# EPICS substitutions: mc1/GalilTestApp/Db/galil_digital_ports.substitutions
# Description:
# digital/binary port substitution file.
#
# This library is free software; you can redistribute it and/or
# modify it under the terms of the GNU Lesser General Public
# Licence as published by the Free Software Foundation; either
# version 2.1 of the Licence, or (at your option) any later version.
#
# This library is distributed in the hope that it will be useful,
# but WITHOUT ANY WARRANTY; without even the implied warranty of
# MERCHANTABILITY or FITNESS FOR A PARTICULAR PURPOSE.  See the GNU
# Lesser General Public Licence for more details.
#
# You should have received a copy of the GNU Lesser General Public
# Licence along with this library; if not, write to the Free Software
# Foundation, Inc., 51 Franklin St, Fifth Floor, Boston, MA 02110-1301 USA.
#
# Contact details:
# Mark Clift
# email: padmoz@tpg.com.au

# P    - PV prefix
# R    - Record Name
# PORT - Asyn port name
# BYTE - Hardware byte to read
# MASK - Mask for this bit

# Digital IO naming
# $(P)$(R)<Byte or word num><Type Bo or Bi><Bit>

file "$(GALIL)/GalilSup/Db/galil_digital_in_bit.template"
{
pattern {P,       R,          PORT,  BYTE,  MASK,     ZNAM,  ONAM,  ZSV,        OSV         , DESC		}

# DMC = Digital motor controller
# DMC binary inputs are organized in bytes
	{"Depo{MC:1}",  DI0BI0,  Galil, 0,     0x000001, "Off", "On",  "NO_ALARM", "MAJOR"  , "Disconnect in Pos"}
	{"Depo{MC:1}",  DI0BI1,  Galil, 0,     0x000002, "Off", "On",  "NO_ALARM", "MAJOR" , "Connect Continuity OK"}
	{"Depo{MC:1}",  DI0BI2,  Galil, 0,     0x000004, "Off", "On",  "NO_ALARM", "MAJOR"  , "Hall Sensor 2"}
	{"Depo{MC:1}",  DI0BI3,  Galil, 0,     0x000008, "Off", "On",  "NO_ALARM", "MAJOR"  , "Hall Sensor 1"}
	{"Depo{MC:1}",  DI0BI4,  Galil, 0,     0x000010, "Off", "On",  "NO_ALARM", "MAJOR"  , "Hall Sensor 3"}
	{"Depo{MC:1}",  DI0BI5,  Galil, 0,     0x000020, "Off", "On",  "NO_ALARM", "MAJOR"  , "PLC Y130"}
	{"Depo{MC:1}",  DI0BI6,  Galil, 0,     0x000040, "Off", "On",  "NO_ALARM", "MAJOR"  , "PLC Y131"}
	{"Depo{MC:1}",  DI0BI7,  Galil, 0,     0x000080, "Off", "On",  "NO_ALARM", "MAJOR"  , "PLC Y132"}
}

# P    - PV prefix
# R    - Record Name
# PORT - Asyn port name
# WORD - Hardware word to read
# MASK - Mask for this bit

file "$(GALIL)/GalilSup/Db/galil_digital_out_bit.template"
{
pattern {P,       R,           PORT,  WORD,  MASK,     ZNAM,  ONAM,  ZSV,        OSV         , DESC		}

# DMC binary outputs are organized in 16bit words
	{"Depo{MC:1}",  DO0BO0,   Galil, 0,     0x000001, "Off", "On",  "NO_ALARM", "NO_ALARM"  , "PLC X70"	}
	{"Depo{MC:1}",  DO0BO1,   Galil, 0,     0x000002, "Off", "On",  "NO_ALARM", "NO_ALARM"  , "PLC X71"	}
	{"Depo{MC:1}",  DO0BO2,   Galil, 0,     0x000004, "Off", "On",  "NO_ALARM", "NO_ALARM"  , "PLC X72"	}
	{"Depo{MC:1}",  DO0BO3,   Galil, 0,     0x000008, "Off", "On",  "NO_ALARM", "NO_ALARM"  , "PLC X73"	}
	{"Depo{MC:1}",  DO0BO4,   Galil, 0,     0x000010, "Off", "On",  "NO_ALARM", "NO_ALARM"  , ""	}
	{"Depo{MC:1}",  DO0BO5,   Galil, 0,     0x000020, "Off", "On",  "NO_ALARM", "NO_ALARM"  , ""	}
	{"Depo{MC:1}",  DO0BO6,   Galil, 0,     0x000040, "Off", "On",  "NO_ALARM", "NO_ALARM"  , ""	}
	{"Depo{MC:1}",  DO0BO7,   Galil, 0,     0x000080, "Off", "On",  "NO_ALARM", "NO_ALARM"  , ""	}
}

# end
